{attribute addProperty BoxType "AX2000-B110-0000"}
{attribute addProperty Id "InputsAT %I*Inputs_352C0ED16480OutputsAT %Q*Outputs_39B5897F4860WcStateAT %I*WcState_F855686C1620InfoDataAT %I*InfoData_6C7DEEF988110"}
{attribute addProperty CRC "535255846"}
{attribute addProperty SizeInBites "216"}
{attribute addProperty SizeInBytes "27"}
TYPE AX2000_9B833B5A :
STRUCT
	{attribute addProperty Name "Inputs"}
	Inputs : Inputs_352C0ED1;
	{attribute addProperty Name "Outputs"}
	Outputs : Outputs_39B5897F;
	{attribute addProperty Name "WcState"}
	WcState : WcState_F855686C;
	{attribute addProperty Name "InfoData"}
	InfoData : InfoData_6C7DEEF9;
END_STRUCT
END_TYPE

(* stored: Version 1.2.0.0, ProductVersion 3.1.4024.9
   DUT AX2000_9B833B5A: Id {75586949-aac5-4f73-9df9-630df133f341} *)
